Fanuc TP program (LS listing): BOTTOM001.LS

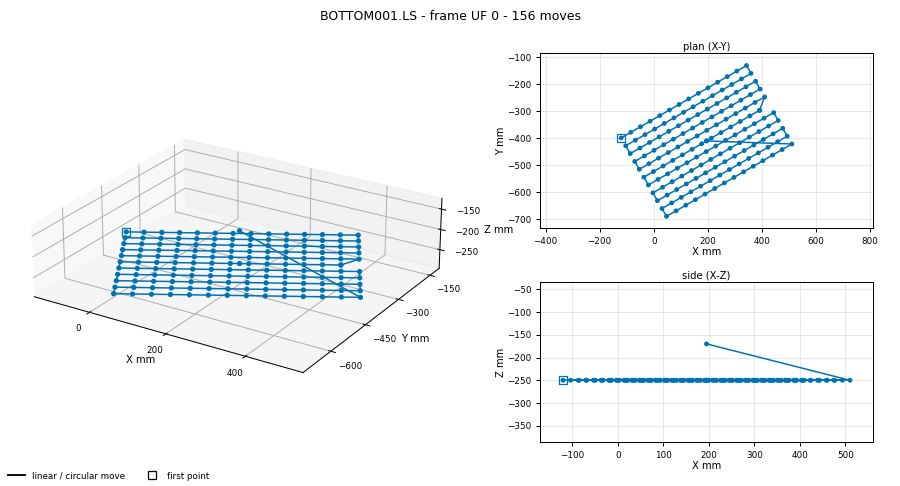
[picture p0: tool path of BOTTOM001.LS in frame UF 0, 156 of 156 moves have a stored position in this frame; points joined in program order, loops and branches not executed]
/PROG  BOTTOM001.LS
/ATTR
OWNER       = MNEDITOR;
COMMENT     = "";
PROG_SIZE   = 636;
CREATE      = DATE 23-01-07  TIME 11:59:14;
MODIFIED    = DATE 23-01-07  TIME 12:02:18;
FILE_NAME   = ;
VERSION     = 0;
LINE_COUNT  = 4;
MEMORY_SIZE = 992;
PROTECT     = READ_WRITE;
TCD:  STACK_SIZE	= 0,
      TASK_PRIORITY	= 50,
      TIME_SLICE	= 0,
      BUSY_LAMP_OFF	= 0,
      ABORT_REQUEST	= 0,
      PAUSE_REQUEST	= 0;
DEFAULT_GROUP	= 1,*,*,*,*;
CONTROL_CODE	= 00000000 00000000;
/MN
   1:J P[1] 100% FINE    ;
   2:L P[2] 100mm/sec CNT0    ;
   3:L P[3] 100mm/sec CNT0    ;
   4:L P[4] 100mm/sec CNT0    ;
   5:L P[5] 100mm/sec CNT0    ;
   6:L P[6] 100mm/sec CNT0    ;
   7:L P[7] 100mm/sec CNT0    ;
   8:L P[8] 100mm/sec CNT0    ;
   9:L P[9] 100mm/sec CNT0    ;
   10:L P[10] 100mm/sec CNT0    ;
   11:L P[11] 100mm/sec CNT0    ;
   12:L P[12] 100mm/sec CNT0    ;
   13:L P[13] 100mm/sec CNT0    ;
   14:L P[14] 100mm/sec CNT0    ;
   15:L P[15] 100mm/sec CNT0    ;
   16:L P[16] 100mm/sec CNT0    ;
   17:L P[17] 100mm/sec CNT0    ;
   18:L P[18] 100mm/sec CNT0    ;
   19:L P[19] 100mm/sec CNT0    ;
   20:L P[20] 100mm/sec CNT0    ;
   21:L P[21] 100mm/sec CNT0    ;
   22:L P[22] 100mm/sec CNT0    ;
   23:L P[23] 100mm/sec CNT0    ;
   24:L P[24] 100mm/sec CNT0    ;
   25:L P[25] 100mm/sec CNT0    ;
   26:L P[26] 100mm/sec CNT0    ;
   27:L P[27] 100mm/sec CNT0    ;
   28:L P[28] 100mm/sec CNT0    ;
   29:L P[29] 100mm/sec CNT0    ;
   30:L P[30] 100mm/sec CNT0    ;
   31:L P[31] 100mm/sec CNT0    ;
   32:L P[32] 100mm/sec CNT0    ;
   33:L P[33] 100mm/sec CNT0    ;
   34:L P[34] 100mm/sec CNT0    ;
   35:L P[35] 100mm/sec CNT0    ;
   36:L P[36] 100mm/sec CNT0    ;
   37:L P[37] 100mm/sec CNT0    ;
   38:L P[38] 100mm/sec CNT0    ;
   39:L P[39] 100mm/sec CNT0    ;
   40:L P[40] 100mm/sec CNT0    ;
   41:L P[41] 100mm/sec CNT0    ;
   42:L P[42] 100mm/sec CNT0    ;
   43:L P[43] 100mm/sec CNT0    ;
   44:L P[44] 100mm/sec CNT0    ;
   45:L P[45] 100mm/sec CNT0    ;
   46:L P[46] 100mm/sec CNT0    ;
   47:L P[47] 100mm/sec CNT0    ;
   48:L P[48] 100mm/sec CNT0    ;
   49:L P[49] 100mm/sec CNT0    ;
   50:L P[50] 100mm/sec CNT0    ;
   51:L P[51] 100mm/sec CNT0    ;
   52:L P[52] 100mm/sec CNT0    ;
   53:L P[53] 100mm/sec CNT0    ;
   54:L P[54] 100mm/sec CNT0    ;
   55:L P[55] 100mm/sec CNT0    ;
   56:L P[56] 100mm/sec CNT0    ;
   57:L P[57] 100mm/sec CNT0    ;
   58:L P[58] 100mm/sec CNT0    ;
   59:L P[59] 100mm/sec CNT0    ;
   60:L P[60] 100mm/sec CNT0    ;
   61:L P[61] 100mm/sec CNT0    ;
   62:L P[62] 100mm/sec CNT0    ;
   63:L P[63] 100mm/sec CNT0    ;
   64:L P[64] 100mm/sec CNT0    ;
   65:L P[65] 100mm/sec CNT0    ;
   66:L P[66] 100mm/sec CNT0    ;
   67:L P[67] 100mm/sec CNT0    ;
   68:L P[68] 100mm/sec CNT0    ;
   69:L P[69] 100mm/sec CNT0    ;
   70:L P[70] 100mm/sec CNT0    ;
   71:L P[71] 100mm/sec CNT0    ;
   72:L P[72] 100mm/sec CNT0    ;
   73:L P[73] 100mm/sec CNT0    ;
   74:L P[74] 100mm/sec CNT0    ;
   75:L P[75] 100mm/sec CNT0    ;
   76:L P[76] 100mm/sec CNT0    ;
   77:L P[77] 100mm/sec CNT0    ;
   78:L P[78] 100mm/sec CNT0    ;
   79:L P[79] 100mm/sec CNT0    ;
   80:L P[80] 100mm/sec CNT0    ;
   81:L P[81] 100mm/sec CNT0    ;
   82:L P[82] 100mm/sec CNT0    ;
   83:L P[83] 100mm/sec CNT0    ;
   84:L P[84] 100mm/sec CNT0    ;
   85:L P[85] 100mm/sec CNT0    ;
   86:L P[86] 100mm/sec CNT0    ;
   87:L P[87] 100mm/sec CNT0    ;
   88:L P[88] 100mm/sec CNT0    ;
   89:L P[89] 100mm/sec CNT0    ;
   90:L P[90] 100mm/sec CNT0    ;
   91:L P[91] 100mm/sec CNT0    ;
   92:L P[92] 100mm/sec CNT0    ;
   93:L P[93] 100mm/sec CNT0    ;
   94:L P[94] 100mm/sec CNT0    ;
   95:L P[95] 100mm/sec CNT0    ;
   96:L P[96] 100mm/sec CNT0    ;
   97:L P[97] 100mm/sec CNT0    ;
   98:L P[98] 100mm/sec CNT0    ;
   99:L P[99] 100mm/sec CNT0    ;
   100:L P[100] 100mm/sec CNT0    ;
   101:L P[101] 100mm/sec CNT0    ;
   102:L P[102] 100mm/sec CNT0    ;
   103:L P[103] 100mm/sec CNT0    ;
   104:L P[104] 100mm/sec CNT0    ;
   105:L P[105] 100mm/sec CNT0    ;
   106:L P[106] 100mm/sec CNT0    ;
   107:L P[107] 100mm/sec CNT0    ;
   108:L P[108] 100mm/sec CNT0    ;
   109:L P[109] 100mm/sec CNT0    ;
   110:L P[110] 100mm/sec CNT0    ;
   111:L P[111] 100mm/sec CNT0    ;
   112:L P[112] 100mm/sec CNT0    ;
   113:L P[113] 100mm/sec CNT0    ;
   114:L P[114] 100mm/sec CNT0    ;
   115:L P[115] 100mm/sec CNT0    ;
   116:L P[116] 100mm/sec CNT0    ;
   117:L P[117] 100mm/sec CNT0    ;
   118:L P[118] 100mm/sec CNT0    ;
   119:L P[119] 100mm/sec CNT0    ;
   120:L P[120] 100mm/sec CNT0    ;
   121:L P[121] 100mm/sec CNT0    ;
   122:L P[122] 100mm/sec CNT0    ;
   123:L P[123] 100mm/sec CNT0    ;
   124:L P[124] 100mm/sec CNT0    ;
   125:L P[125] 100mm/sec CNT0    ;
   126:L P[126] 100mm/sec CNT0    ;
   127:L P[127] 100mm/sec CNT0    ;
   128:L P[128] 100mm/sec CNT0    ;
   129:L P[129] 100mm/sec CNT0    ;
   130:L P[130] 100mm/sec CNT0    ;
   131:L P[131] 100mm/sec CNT0    ;
   132:L P[132] 100mm/sec CNT0    ;
   133:L P[133] 100mm/sec CNT0    ;
   134:L P[134] 100mm/sec CNT0    ;
   135:L P[135] 100mm/sec CNT0    ;
   136:L P[136] 100mm/sec CNT0    ;
   137:L P[137] 100mm/sec CNT0    ;
   138:L P[138] 100mm/sec CNT0    ;
   139:L P[139] 100mm/sec CNT0    ;
   140:L P[140] 100mm/sec CNT0    ;
   141:L P[141] 100mm/sec CNT0    ;
   142:L P[142] 100mm/sec CNT0    ;
   143:L P[143] 100mm/sec CNT0    ;
   144:L P[144] 100mm/sec CNT0    ;
   145:L P[145] 100mm/sec CNT0    ;
   146:L P[146] 100mm/sec CNT0    ;
   147:L P[147] 100mm/sec CNT0    ;
   148:L P[148] 100mm/sec CNT0    ;
   149:L P[149] 100mm/sec CNT0    ;
   150:L P[150] 100mm/sec CNT0    ;
   151:L P[151] 100mm/sec CNT0    ;
   152:L P[152] 100mm/sec CNT0    ;
   153:L P[153] 100mm/sec CNT0    ;
   154:L P[154] 100mm/sec CNT0    ;
   155:L P[155] 100mm/sec CNT0    ;
   156:L P[156] 100mm/sec CNT0    ;
/POS
P[1]{
   GP1:
	UF : 0, UT : 6,		CONFIG : 'N U T, 0, 0, 0',
	X =  -120.438  mm,	Y =   -398.694  mm,	Z =   -250.000  mm,
	W =  90.000 deg,	P =   0.000 deg,	R =   90.000 deg
};
P[2]{
   GP1:
	UF : 0, UT : 6,		CONFIG : 'N U T, 0, 0, 0',
	X =  -84.795  mm,	Y =   -378.115  mm,	Z =   -250.000  mm,
	W =  90.000 deg,	P =   0.000 deg,	R =   90.000 deg
};
P[3]{
   GP1:
	UF : 0, UT : 6,		CONFIG : 'N U T, 0, 0, 0',
	X =  -49.153  mm,	Y =   -357.535  mm,	Z =   -250.000  mm,
	W =  90.000 deg,	P =   0.000 deg,	R =   90.000 deg
};
P[4]{
   GP1:
	UF : 0, UT : 6,		CONFIG : 'N U T, 0, 0, 0',
	X =  -13.511  mm,	Y =   -336.956  mm,	Z =   -250.000  mm,
	W =  90.000 deg,	P =   0.000 deg,	R =   90.000 deg
};
P[5]{
   GP1:
	UF : 0, UT : 6,		CONFIG : 'N U T, 0, 0, 0',
	X =  22.131  mm,	Y =   -316.376  mm,	Z =   -250.000  mm,
	W =  90.000 deg,	P =   0.000 deg,	R =   90.000 deg
};
P[6]{
   GP1:
	UF : 0, UT : 6,		CONFIG : 'N U T, 0, 0, 0',
	X =  57.773  mm,	Y =   -295.797  mm,	Z =   -250.000  mm,
	W =  90.000 deg,	P =   0.000 deg,	R =   90.000 deg
};
P[7]{
   GP1:
	UF : 0, UT : 6,		CONFIG : 'N U T, 0, 0, 0',
	X =  93.415  mm,	Y =   -275.217  mm,	Z =   -250.000  mm,
	W =  90.000 deg,	P =   0.000 deg,	R =   90.000 deg
};
P[8]{
   GP1:
	UF : 0, UT : 6,		CONFIG : 'N U T, 0, 0, 0',
	X =  129.058  mm,	Y =   -254.638  mm,	Z =   -250.000  mm,
	W =  90.000 deg,	P =   0.000 deg,	R =   90.000 deg
};
P[9]{
   GP1:
	UF : 0, UT : 6,		CONFIG : 'N U T, 0, 0, 0',
	X =  164.700  mm,	Y =   -234.059  mm,	Z =   -250.000  mm,
	W =  90.000 deg,	P =   0.000 deg,	R =   90.000 deg
};
P[10]{
   GP1:
	UF : 0, UT : 6,		CONFIG : 'N U T, 0, 0, 0',
	X =  200.342  mm,	Y =   -213.479  mm,	Z =   -250.000  mm,
	W =  90.000 deg,	P =   0.000 deg,	R =   90.000 deg
};
P[11]{
   GP1:
	UF : 0, UT : 6,		CONFIG : 'N U T, 0, 0, 0',
	X =  235.984  mm,	Y =   -192.900  mm,	Z =   -250.000  mm,
	W =  90.000 deg,	P =   0.000 deg,	R =   90.000 deg
};
P[12]{
   GP1:
	UF : 0, UT : 6,		CONFIG : 'N U T, 0, 0, 0',
	X =  271.626  mm,	Y =   -172.320  mm,	Z =   -250.000  mm,
	W =  90.000 deg,	P =   0.000 deg,	R =   90.000 deg
};
P[13]{
   GP1:
	UF : 0, UT : 6,		CONFIG : 'N U T, 0, 0, 0',
	X =  307.268  mm,	Y =   -151.741  mm,	Z =   -250.000  mm,
	W =  90.000 deg,	P =   0.000 deg,	R =   90.000 deg
};
P[14]{
   GP1:
	UF : 0, UT : 6,		CONFIG : 'N U T, 0, 0, 0',
	X =  342.911  mm,	Y =   -131.161  mm,	Z =   -250.000  mm,
	W =  90.000 deg,	P =   0.000 deg,	R =   90.000 deg
};
P[15]{
   GP1:
	UF : 0, UT : 6,		CONFIG : 'N U T, 0, 0, 0',
	X =  359.663  mm,	Y =   -160.176  mm,	Z =   -250.000  mm,
	W =  90.000 deg,	P =   0.000 deg,	R =   90.000 deg
};
P[16]{
   GP1:
	UF : 0, UT : 6,		CONFIG : 'N U T, 0, 0, 0',
	X =  324.021  mm,	Y =   -180.755  mm,	Z =   -250.000  mm,
	W =  90.000 deg,	P =   0.000 deg,	R =   90.000 deg
};
P[17]{
   GP1:
	UF : 0, UT : 6,		CONFIG : 'N U T, 0, 0, 0',
	X =  288.379  mm,	Y =   -201.335  mm,	Z =   -250.000  mm,
	W =  90.000 deg,	P =   0.000 deg,	R =   90.000 deg
};
P[18]{
   GP1:
	UF : 0, UT : 6,		CONFIG : 'N U T, 0, 0, 0',
	X =  252.737  mm,	Y =   -221.914  mm,	Z =   -250.000  mm,
	W =  90.000 deg,	P =   0.000 deg,	R =   90.000 deg
};
P[19]{
   GP1:
	UF : 0, UT : 6,		CONFIG : 'N U T, 0, 0, 0',
	X =  217.095  mm,	Y =   -242.493  mm,	Z =   -250.000  mm,
	W =  90.000 deg,	P =   0.000 deg,	R =   90.000 deg
};
P[20]{
   GP1:
	UF : 0, UT : 6,		CONFIG : 'N U T, 0, 0, 0',
	X =  181.452  mm,	Y =   -263.073  mm,	Z =   -250.000  mm,
	W =  90.000 deg,	P =   0.000 deg,	R =   90.000 deg
};
P[21]{
   GP1:
	UF : 0, UT : 6,		CONFIG : 'N U T, 0, 0, 0',
	X =  145.810  mm,	Y =   -283.652  mm,	Z =   -250.000  mm,
	W =  90.000 deg,	P =   0.000 deg,	R =   90.000 deg
};
P[22]{
   GP1:
	UF : 0, UT : 6,		CONFIG : 'N U T, 0, 0, 0',
	X =  110.168  mm,	Y =   -304.232  mm,	Z =   -250.000  mm,
	W =  90.000 deg,	P =   0.000 deg,	R =   90.000 deg
};
P[23]{
   GP1:
	UF : 0, UT : 6,		CONFIG : 'N U T, 0, 0, 0',
	X =  74.526  mm,	Y =   -324.811  mm,	Z =   -250.000  mm,
	W =  90.000 deg,	P =   0.000 deg,	R =   90.000 deg
};
P[24]{
   GP1:
	UF : 0, UT : 6,		CONFIG : 'N U T, 0, 0, 0',
	X =  38.884  mm,	Y =   -345.391  mm,	Z =   -250.000  mm,
	W =  90.000 deg,	P =   0.000 deg,	R =   90.000 deg
};
P[25]{
   GP1:
	UF : 0, UT : 6,		CONFIG : 'N U T, 0, 0, 0',
	X =  3.242  mm,	Y =   -365.970  mm,	Z =   -250.000  mm,
	W =  90.000 deg,	P =   0.000 deg,	R =   90.000 deg
};
P[26]{
   GP1:
	UF : 0, UT : 6,		CONFIG : 'N U T, 0, 0, 0',
	X =  -32.401  mm,	Y =   -386.550  mm,	Z =   -250.000  mm,
	W =  90.000 deg,	P =   0.000 deg,	R =   90.000 deg
};
P[27]{
   GP1:
	UF : 0, UT : 6,		CONFIG : 'N U T, 0, 0, 0',
	X =  -68.043  mm,	Y =   -407.129  mm,	Z =   -250.000  mm,
	W =  90.000 deg,	P =   0.000 deg,	R =   90.000 deg
};
P[28]{
   GP1:
	UF : 0, UT : 6,		CONFIG : 'N U T, 0, 0, 0',
	X =  -103.685  mm,	Y =   -427.709  mm,	Z =   -250.000  mm,
	W =  90.000 deg,	P =   0.000 deg,	R =   90.000 deg
};
P[29]{
   GP1:
	UF : 0, UT : 6,		CONFIG : 'N U T, 0, 0, 0',
	X =  -86.932  mm,	Y =   -456.723  mm,	Z =   -250.000  mm,
	W =  90.000 deg,	P =   0.000 deg,	R =   90.000 deg
};
P[30]{
   GP1:
	UF : 0, UT : 6,		CONFIG : 'N U T, 0, 0, 0',
	X =  -51.290  mm,	Y =   -436.144  mm,	Z =   -250.000  mm,
	W =  90.000 deg,	P =   0.000 deg,	R =   90.000 deg
};
P[31]{
   GP1:
	UF : 0, UT : 6,		CONFIG : 'N U T, 0, 0, 0',
	X =  -15.648  mm,	Y =   -415.564  mm,	Z =   -250.000  mm,
	W =  90.000 deg,	P =   0.000 deg,	R =   90.000 deg
};
P[32]{
   GP1:
	UF : 0, UT : 6,		CONFIG : 'N U T, 0, 0, 0',
	X =  19.994  mm,	Y =   -394.985  mm,	Z =   -250.000  mm,
	W =  90.000 deg,	P =   0.000 deg,	R =   90.000 deg
};
P[33]{
   GP1:
	UF : 0, UT : 6,		CONFIG : 'N U T, 0, 0, 0',
	X =  55.636  mm,	Y =   -374.405  mm,	Z =   -250.000  mm,
	W =  90.000 deg,	P =   0.000 deg,	R =   90.000 deg
};
P[34]{
   GP1:
	UF : 0, UT : 6,		CONFIG : 'N U T, 0, 0, 0',
	X =  91.279  mm,	Y =   -353.826  mm,	Z =   -250.000  mm,
	W =  90.000 deg,	P =   0.000 deg,	R =   90.000 deg
};
P[35]{
   GP1:
	UF : 0, UT : 6,		CONFIG : 'N U T, 0, 0, 0',
	X =  126.921  mm,	Y =   -333.246  mm,	Z =   -250.000  mm,
	W =  90.000 deg,	P =   0.000 deg,	R =   90.000 deg
};
P[36]{
   GP1:
	UF : 0, UT : 6,		CONFIG : 'N U T, 0, 0, 0',
	X =  162.563  mm,	Y =   -312.667  mm,	Z =   -250.000  mm,
	W =  90.000 deg,	P =   0.000 deg,	R =   90.000 deg
};
P[37]{
   GP1:
	UF : 0, UT : 6,		CONFIG : 'N U T, 0, 0, 0',
	X =  198.205  mm,	Y =   -292.087  mm,	Z =   -250.000  mm,
	W =  90.000 deg,	P =   0.000 deg,	R =   90.000 deg
};
P[38]{
   GP1:
	UF : 0, UT : 6,		CONFIG : 'N U T, 0, 0, 0',
	X =  233.847  mm,	Y =   -271.508  mm,	Z =   -250.000  mm,
	W =  90.000 deg,	P =   0.000 deg,	R =   90.000 deg
};
P[39]{
   GP1:
	UF : 0, UT : 6,		CONFIG : 'N U T, 0, 0, 0',
	X =  269.490  mm,	Y =   -250.928  mm,	Z =   -250.000  mm,
	W =  90.000 deg,	P =   0.000 deg,	R =   90.000 deg
};
P[40]{
   GP1:
	UF : 0, UT : 6,		CONFIG : 'N U T, 0, 0, 0',
	X =  305.132  mm,	Y =   -230.349  mm,	Z =   -250.000  mm,
	W =  90.000 deg,	P =   0.000 deg,	R =   90.000 deg
};
P[41]{
   GP1:
	UF : 0, UT : 6,		CONFIG : 'N U T, 0, 0, 0',
	X =  340.774  mm,	Y =   -209.769  mm,	Z =   -250.000  mm,
	W =  90.000 deg,	P =   0.000 deg,	R =   90.000 deg
};
P[42]{
   GP1:
	UF : 0, UT : 6,		CONFIG : 'N U T, 0, 0, 0',
	X =  376.416  mm,	Y =   -189.190  mm,	Z =   -250.000  mm,
	W =  90.000 deg,	P =   0.000 deg,	R =   90.000 deg
};
P[43]{
   GP1:
	UF : 0, UT : 6,		CONFIG : 'N U T, 0, 0, 0',
	X =  393.169  mm,	Y =   -218.204  mm,	Z =   -250.000  mm,
	W =  90.000 deg,	P =   0.000 deg,	R =   90.000 deg
};
P[44]{
   GP1:
	UF : 0, UT : 6,		CONFIG : 'N U T, 0, 0, 0',
	X =  357.527  mm,	Y =   -238.784  mm,	Z =   -250.000  mm,
	W =  90.000 deg,	P =   0.000 deg,	R =   90.000 deg
};
P[45]{
   GP1:
	UF : 0, UT : 6,		CONFIG : 'N U T, 0, 0, 0',
	X =  321.884  mm,	Y =   -259.363  mm,	Z =   -250.000  mm,
	W =  90.000 deg,	P =   0.000 deg,	R =   90.000 deg
};
P[46]{
   GP1:
	UF : 0, UT : 6,		CONFIG : 'N U T, 0, 0, 0',
	X =  286.242  mm,	Y =   -279.943  mm,	Z =   -250.000  mm,
	W =  90.000 deg,	P =   0.000 deg,	R =   90.000 deg
};
P[47]{
   GP1:
	UF : 0, UT : 6,		CONFIG : 'N U T, 0, 0, 0',
	X =  250.600  mm,	Y =   -300.522  mm,	Z =   -250.000  mm,
	W =  90.000 deg,	P =   0.000 deg,	R =   90.000 deg
};
P[48]{
   GP1:
	UF : 0, UT : 6,		CONFIG : 'N U T, 0, 0, 0',
	X =  214.958  mm,	Y =   -321.102  mm,	Z =   -250.000  mm,
	W =  90.000 deg,	P =   0.000 deg,	R =   90.000 deg
};
P[49]{
   GP1:
	UF : 0, UT : 6,		CONFIG : 'N U T, 0, 0, 0',
	X =  179.316  mm,	Y =   -341.681  mm,	Z =   -250.000  mm,
	W =  90.000 deg,	P =   0.000 deg,	R =   90.000 deg
};
P[50]{
   GP1:
	UF : 0, UT : 6,		CONFIG : 'N U T, 0, 0, 0',
	X =  143.674  mm,	Y =   -362.261  mm,	Z =   -250.000  mm,
	W =  90.000 deg,	P =   0.000 deg,	R =   90.000 deg
};
P[51]{
   GP1:
	UF : 0, UT : 6,		CONFIG : 'N U T, 0, 0, 0',
	X =  108.031  mm,	Y =   -382.840  mm,	Z =   -250.000  mm,
	W =  90.000 deg,	P =   0.000 deg,	R =   90.000 deg
};
P[52]{
   GP1:
	UF : 0, UT : 6,		CONFIG : 'N U T, 0, 0, 0',
	X =  72.389  mm,	Y =   -403.420  mm,	Z =   -250.000  mm,
	W =  90.000 deg,	P =   0.000 deg,	R =   90.000 deg
};
P[53]{
   GP1:
	UF : 0, UT : 6,		CONFIG : 'N U T, 0, 0, 0',
	X =  36.747  mm,	Y =   -423.999  mm,	Z =   -250.000  mm,
	W =  90.000 deg,	P =   0.000 deg,	R =   90.000 deg
};
P[54]{
   GP1:
	UF : 0, UT : 6,		CONFIG : 'N U T, 0, 0, 0',
	X =  1.105  mm,	Y =   -444.579  mm,	Z =   -250.000  mm,
	W =  90.000 deg,	P =   0.000 deg,	R =   90.000 deg
};
P[55]{
   GP1:
	UF : 0, UT : 6,		CONFIG : 'N U T, 0, 0, 0',
	X =  -34.537  mm,	Y =   -465.158  mm,	Z =   -250.000  mm,
	W =  90.000 deg,	P =   0.000 deg,	R =   90.000 deg
};
P[56]{
   GP1:
	UF : 0, UT : 6,		CONFIG : 'N U T, 0, 0, 0',
	X =  -70.180  mm,	Y =   -485.738  mm,	Z =   -250.000  mm,
	W =  90.000 deg,	P =   0.000 deg,	R =   90.000 deg
};
P[57]{
   GP1:
	UF : 0, UT : 6,		CONFIG : 'N U T, 0, 0, 0',
	X =  -53.427  mm,	Y =   -514.752  mm,	Z =   -250.000  mm,
	W =  90.000 deg,	P =   0.000 deg,	R =   90.000 deg
};
P[58]{
   GP1:
	UF : 0, UT : 6,		CONFIG : 'N U T, 0, 0, 0',
	X =  -17.785  mm,	Y =   -494.173  mm,	Z =   -250.000  mm,
	W =  90.000 deg,	P =   0.000 deg,	R =   90.000 deg
};
P[59]{
   GP1:
	UF : 0, UT : 6,		CONFIG : 'N U T, 0, 0, 0',
	X =  17.858  mm,	Y =   -473.593  mm,	Z =   -250.000  mm,
	W =  90.000 deg,	P =   0.000 deg,	R =   90.000 deg
};
P[60]{
   GP1:
	UF : 0, UT : 6,		CONFIG : 'N U T, 0, 0, 0',
	X =  53.500  mm,	Y =   -453.014  mm,	Z =   -250.000  mm,
	W =  90.000 deg,	P =   0.000 deg,	R =   90.000 deg
};
P[61]{
   GP1:
	UF : 0, UT : 6,		CONFIG : 'N U T, 0, 0, 0',
	X =  89.142  mm,	Y =   -432.434  mm,	Z =   -250.000  mm,
	W =  90.000 deg,	P =   0.000 deg,	R =   90.000 deg
};
P[62]{
   GP1:
	UF : 0, UT : 6,		CONFIG : 'N U T, 0, 0, 0',
	X =  124.784  mm,	Y =   -411.855  mm,	Z =   -250.000  mm,
	W =  90.000 deg,	P =   0.000 deg,	R =   90.000 deg
};
P[63]{
   GP1:
	UF : 0, UT : 6,		CONFIG : 'N U T, 0, 0, 0',
	X =  160.426  mm,	Y =   -391.275  mm,	Z =   -250.000  mm,
	W =  90.000 deg,	P =   0.000 deg,	R =   90.000 deg
};
P[64]{
   GP1:
	UF : 0, UT : 6,		CONFIG : 'N U T, 0, 0, 0',
	X =  196.068  mm,	Y =   -370.696  mm,	Z =   -250.000  mm,
	W =  90.000 deg,	P =   0.000 deg,	R =   90.000 deg
};
P[65]{
   GP1:
	UF : 0, UT : 6,		CONFIG : 'N U T, 0, 0, 0',
	X =  231.711  mm,	Y =   -350.116  mm,	Z =   -250.000  mm,
	W =  90.000 deg,	P =   0.000 deg,	R =   90.000 deg
};
P[66]{
   GP1:
	UF : 0, UT : 6,		CONFIG : 'N U T, 0, 0, 0',
	X =  267.353  mm,	Y =   -329.537  mm,	Z =   -250.000  mm,
	W =  90.000 deg,	P =   0.000 deg,	R =   90.000 deg
};
P[67]{
   GP1:
	UF : 0, UT : 6,		CONFIG : 'N U T, 0, 0, 0',
	X =  302.995  mm,	Y =   -308.957  mm,	Z =   -250.000  mm,
	W =  90.000 deg,	P =   0.000 deg,	R =   90.000 deg
};
P[68]{
   GP1:
	UF : 0, UT : 6,		CONFIG : 'N U T, 0, 0, 0',
	X =  338.637  mm,	Y =   -288.378  mm,	Z =   -250.000  mm,
	W =  90.000 deg,	P =   0.000 deg,	R =   90.000 deg
};
P[69]{
   GP1:
	UF : 0, UT : 6,		CONFIG : 'N U T, 0, 0, 0',
	X =  374.279  mm,	Y =   -267.798  mm,	Z =   -250.000  mm,
	W =  90.000 deg,	P =   0.000 deg,	R =   90.000 deg
};
P[70]{
   GP1:
	UF : 0, UT : 6,		CONFIG : 'N U T, 0, 0, 0',
	X =  409.921  mm,	Y =   -247.219  mm,	Z =   -250.000  mm,
	W =  90.000 deg,	P =   0.000 deg,	R =   90.000 deg
};
P[71]{
   GP1:
	UF : 0, UT : 6,		CONFIG : 'N U T, 0, 0, 0',
	X =  391.032  mm,	Y =   -296.813  mm,	Z =   -250.000  mm,
	W =  90.000 deg,	P =   0.000 deg,	R =   90.000 deg
};
P[72]{
   GP1:
	UF : 0, UT : 6,		CONFIG : 'N U T, 0, 0, 0',
	X =  391.032  mm,	Y =   -296.813  mm,	Z =   -250.000  mm,
	W =  90.000 deg,	P =   0.000 deg,	R =   90.000 deg
};
P[73]{
   GP1:
	UF : 0, UT : 6,		CONFIG : 'N U T, 0, 0, 0',
	X =  355.390  mm,	Y =   -317.392  mm,	Z =   -250.000  mm,
	W =  90.000 deg,	P =   0.000 deg,	R =   90.000 deg
};
P[74]{
   GP1:
	UF : 0, UT : 6,		CONFIG : 'N U T, 0, 0, 0',
	X =  319.748  mm,	Y =   -337.972  mm,	Z =   -250.000  mm,
	W =  90.000 deg,	P =   0.000 deg,	R =   90.000 deg
};
P[75]{
   GP1:
	UF : 0, UT : 6,		CONFIG : 'N U T, 0, 0, 0',
	X =  284.105  mm,	Y =   -358.551  mm,	Z =   -250.000  mm,
	W =  90.000 deg,	P =   0.000 deg,	R =   90.000 deg
};
P[76]{
   GP1:
	UF : 0, UT : 6,		CONFIG : 'N U T, 0, 0, 0',
	X =  248.463  mm,	Y =   -379.131  mm,	Z =   -250.000  mm,
	W =  90.000 deg,	P =   0.000 deg,	R =   90.000 deg
};
P[77]{
   GP1:
	UF : 0, UT : 6,		CONFIG : 'N U T, 0, 0, 0',
	X =  212.821  mm,	Y =   -399.710  mm,	Z =   -250.000  mm,
	W =  90.000 deg,	P =   0.000 deg,	R =   90.000 deg
};
P[78]{
   GP1:
	UF : 0, UT : 6,		CONFIG : 'N U T, 0, 0, 0',
	X =  195.000  mm,	Y =   -410.000  mm,	Z =   -250.000  mm,
	W =  90.000 deg,	P =   0.000 deg,	R =   90.000 deg
};
P[79]{
   GP1:
	UF : 0, UT : 6,		CONFIG : 'N U T, 0, 0, 0',
	X =  177.179  mm,	Y =   -420.290  mm,	Z =   -250.000  mm,
	W =  90.000 deg,	P =   0.000 deg,	R =   90.000 deg
};
P[80]{
   GP1:
	UF : 0, UT : 6,		CONFIG : 'N U T, 0, 0, 0',
	X =  141.537  mm,	Y =   -440.869  mm,	Z =   -250.000  mm,
	W =  90.000 deg,	P =   0.000 deg,	R =   90.000 deg
};
P[81]{
   GP1:
	UF : 0, UT : 6,		CONFIG : 'N U T, 0, 0, 0',
	X =  105.895  mm,	Y =   -461.449  mm,	Z =   -250.000  mm,
	W =  90.000 deg,	P =   0.000 deg,	R =   90.000 deg
};
P[82]{
   GP1:
	UF : 0, UT : 6,		CONFIG : 'N U T, 0, 0, 0',
	X =  70.252  mm,	Y =   -482.028  mm,	Z =   -250.000  mm,
	W =  90.000 deg,	P =   0.000 deg,	R =   90.000 deg
};
P[83]{
   GP1:
	UF : 0, UT : 6,		CONFIG : 'N U T, 0, 0, 0',
	X =  34.610  mm,	Y =   -502.608  mm,	Z =   -250.000  mm,
	W =  90.000 deg,	P =   0.000 deg,	R =   90.000 deg
};
P[84]{
   GP1:
	UF : 0, UT : 6,		CONFIG : 'N U T, 0, 0, 0',
	X =  -1.032  mm,	Y =   -523.187  mm,	Z =   -250.000  mm,
	W =  90.000 deg,	P =   0.000 deg,	R =   90.000 deg
};
P[85]{
   GP1:
	UF : 0, UT : 6,		CONFIG : 'N U T, 0, 0, 0',
	X =  -36.674  mm,	Y =   -543.767  mm,	Z =   -250.000  mm,
	W =  90.000 deg,	P =   0.000 deg,	R =   90.000 deg
};
P[86]{
   GP1:
	UF : 0, UT : 6,		CONFIG : 'N U T, 0, 0, 0',
	X =  -19.921  mm,	Y =   -572.781  mm,	Z =   -250.000  mm,
	W =  90.000 deg,	P =   0.000 deg,	R =   90.000 deg
};
P[87]{
   GP1:
	UF : 0, UT : 6,		CONFIG : 'N U T, 0, 0, 0',
	X =  15.721  mm,	Y =   -552.202  mm,	Z =   -250.000  mm,
	W =  90.000 deg,	P =   0.000 deg,	R =   90.000 deg
};
P[88]{
   GP1:
	UF : 0, UT : 6,		CONFIG : 'N U T, 0, 0, 0',
	X =  51.363  mm,	Y =   -531.622  mm,	Z =   -250.000  mm,
	W =  90.000 deg,	P =   0.000 deg,	R =   90.000 deg
};
P[89]{
   GP1:
	UF : 0, UT : 6,		CONFIG : 'N U T, 0, 0, 0',
	X =  87.005  mm,	Y =   -511.043  mm,	Z =   -250.000  mm,
	W =  90.000 deg,	P =   0.000 deg,	R =   90.000 deg
};
P[90]{
   GP1:
	UF : 0, UT : 6,		CONFIG : 'N U T, 0, 0, 0',
	X =  122.647  mm,	Y =   -490.463  mm,	Z =   -250.000  mm,
	W =  90.000 deg,	P =   0.000 deg,	R =   90.000 deg
};
P[91]{
   GP1:
	UF : 0, UT : 6,		CONFIG : 'N U T, 0, 0, 0',
	X =  158.289  mm,	Y =   -469.884  mm,	Z =   -250.000  mm,
	W =  90.000 deg,	P =   0.000 deg,	R =   90.000 deg
};
P[92]{
   GP1:
	UF : 0, UT : 6,		CONFIG : 'N U T, 0, 0, 0',
	X =  193.932  mm,	Y =   -449.304  mm,	Z =   -250.000  mm,
	W =  90.000 deg,	P =   0.000 deg,	R =   90.000 deg
};
P[93]{
   GP1:
	UF : 0, UT : 6,		CONFIG : 'N U T, 0, 0, 0',
	X =  229.574  mm,	Y =   -428.725  mm,	Z =   -250.000  mm,
	W =  90.000 deg,	P =   0.000 deg,	R =   90.000 deg
};
P[94]{
   GP1:
	UF : 0, UT : 6,		CONFIG : 'N U T, 0, 0, 0',
	X =  265.216  mm,	Y =   -408.145  mm,	Z =   -250.000  mm,
	W =  90.000 deg,	P =   0.000 deg,	R =   90.000 deg
};
P[95]{
   GP1:
	UF : 0, UT : 6,		CONFIG : 'N U T, 0, 0, 0',
	X =  300.858  mm,	Y =   -387.566  mm,	Z =   -250.000  mm,
	W =  90.000 deg,	P =   0.000 deg,	R =   90.000 deg
};
P[96]{
   GP1:
	UF : 0, UT : 6,		CONFIG : 'N U T, 0, 0, 0',
	X =  336.500  mm,	Y =   -366.986  mm,	Z =   -250.000  mm,
	W =  90.000 deg,	P =   0.000 deg,	R =   90.000 deg
};
P[97]{
   GP1:
	UF : 0, UT : 6,		CONFIG : 'N U T, 0, 0, 0',
	X =  372.142  mm,	Y =   -346.407  mm,	Z =   -250.000  mm,
	W =  90.000 deg,	P =   0.000 deg,	R =   90.000 deg
};
P[98]{
   GP1:
	UF : 0, UT : 6,		CONFIG : 'N U T, 0, 0, 0',
	X =  407.785  mm,	Y =   -325.827  mm,	Z =   -250.000  mm,
	W =  90.000 deg,	P =   0.000 deg,	R =   90.000 deg
};
P[99]{
   GP1:
	UF : 0, UT : 6,		CONFIG : 'N U T, 0, 0, 0',
	X =  443.427  mm,	Y =   -305.248  mm,	Z =   -250.000  mm,
	W =  90.000 deg,	P =   0.000 deg,	R =   90.000 deg
};
P[100]{
   GP1:
	UF : 0, UT : 6,		CONFIG : 'N U T, 0, 0, 0',
	X =  460.180  mm,	Y =   -334.262  mm,	Z =   -250.000  mm,
	W =  90.000 deg,	P =   0.000 deg,	R =   90.000 deg
};
P[101]{
   GP1:
	UF : 0, UT : 6,		CONFIG : 'N U T, 0, 0, 0',
	X =  424.537  mm,	Y =   -354.842  mm,	Z =   -250.000  mm,
	W =  90.000 deg,	P =   0.000 deg,	R =   90.000 deg
};
P[102]{
   GP1:
	UF : 0, UT : 6,		CONFIG : 'N U T, 0, 0, 0',
	X =  388.895  mm,	Y =   -375.421  mm,	Z =   -250.000  mm,
	W =  90.000 deg,	P =   0.000 deg,	R =   90.000 deg
};
P[103]{
   GP1:
	UF : 0, UT : 6,		CONFIG : 'N U T, 0, 0, 0',
	X =  353.253  mm,	Y =   -396.001  mm,	Z =   -250.000  mm,
	W =  90.000 deg,	P =   0.000 deg,	R =   90.000 deg
};
P[104]{
   GP1:
	UF : 0, UT : 6,		CONFIG : 'N U T, 0, 0, 0',
	X =  317.611  mm,	Y =   -416.580  mm,	Z =   -250.000  mm,
	W =  90.000 deg,	P =   0.000 deg,	R =   90.000 deg
};
P[105]{
   GP1:
	UF : 0, UT : 6,		CONFIG : 'N U T, 0, 0, 0',
	X =  281.969  mm,	Y =   -437.160  mm,	Z =   -250.000  mm,
	W =  90.000 deg,	P =   0.000 deg,	R =   90.000 deg
};
P[106]{
   GP1:
	UF : 0, UT : 6,		CONFIG : 'N U T, 0, 0, 0',
	X =  246.326  mm,	Y =   -457.739  mm,	Z =   -250.000  mm,
	W =  90.000 deg,	P =   0.000 deg,	R =   90.000 deg
};
P[107]{
   GP1:
	UF : 0, UT : 6,		CONFIG : 'N U T, 0, 0, 0',
	X =  210.684  mm,	Y =   -478.319  mm,	Z =   -250.000  mm,
	W =  90.000 deg,	P =   0.000 deg,	R =   90.000 deg
};
P[108]{
   GP1:
	UF : 0, UT : 6,		CONFIG : 'N U T, 0, 0, 0',
	X =  175.042  mm,	Y =   -498.898  mm,	Z =   -250.000  mm,
	W =  90.000 deg,	P =   0.000 deg,	R =   90.000 deg
};
P[109]{
   GP1:
	UF : 0, UT : 6,		CONFIG : 'N U T, 0, 0, 0',
	X =  139.400  mm,	Y =   -519.478  mm,	Z =   -250.000  mm,
	W =  90.000 deg,	P =   0.000 deg,	R =   90.000 deg
};
P[110]{
   GP1:
	UF : 0, UT : 6,		CONFIG : 'N U T, 0, 0, 0',
	X =  103.758  mm,	Y =   -540.057  mm,	Z =   -250.000  mm,
	W =  90.000 deg,	P =   0.000 deg,	R =   90.000 deg
};
P[111]{
   GP1:
	UF : 0, UT : 6,		CONFIG : 'N U T, 0, 0, 0',
	X =  68.116  mm,	Y =   -560.637  mm,	Z =   -250.000  mm,
	W =  90.000 deg,	P =   0.000 deg,	R =   90.000 deg
};
P[112]{
   GP1:
	UF : 0, UT : 6,		CONFIG : 'N U T, 0, 0, 0',
	X =  32.473  mm,	Y =   -581.216  mm,	Z =   -250.000  mm,
	W =  90.000 deg,	P =   0.000 deg,	R =   90.000 deg
};
P[113]{
   GP1:
	UF : 0, UT : 6,		CONFIG : 'N U T, 0, 0, 0',
	X =  -3.169  mm,	Y =   -601.796  mm,	Z =   -250.000  mm,
	W =  90.000 deg,	P =   0.000 deg,	R =   90.000 deg
};
P[114]{
   GP1:
	UF : 0, UT : 6,		CONFIG : 'N U T, 0, 0, 0',
	X =  13.584  mm,	Y =   -630.810  mm,	Z =   -250.000  mm,
	W =  90.000 deg,	P =   0.000 deg,	R =   90.000 deg
};
P[115]{
   GP1:
	UF : 0, UT : 6,		CONFIG : 'N U T, 0, 0, 0',
	X =  49.226  mm,	Y =   -610.231  mm,	Z =   -250.000  mm,
	W =  90.000 deg,	P =   0.000 deg,	R =   90.000 deg
};
P[116]{
   GP1:
	UF : 0, UT : 6,		CONFIG : 'N U T, 0, 0, 0',
	X =  84.868  mm,	Y =   -589.651  mm,	Z =   -250.000  mm,
	W =  90.000 deg,	P =   0.000 deg,	R =   90.000 deg
};
P[117]{
   GP1:
	UF : 0, UT : 6,		CONFIG : 'N U T, 0, 0, 0',
	X =  120.510  mm,	Y =   -569.072  mm,	Z =   -250.000  mm,
	W =  90.000 deg,	P =   0.000 deg,	R =   90.000 deg
};
P[118]{
   GP1:
	UF : 0, UT : 6,		CONFIG : 'N U T, 0, 0, 0',
	X =  156.153  mm,	Y =   -548.492  mm,	Z =   -250.000  mm,
	W =  90.000 deg,	P =   0.000 deg,	R =   90.000 deg
};
P[119]{
   GP1:
	UF : 0, UT : 6,		CONFIG : 'N U T, 0, 0, 0',
	X =  191.795  mm,	Y =   -527.913  mm,	Z =   -250.000  mm,
	W =  90.000 deg,	P =   0.000 deg,	R =   90.000 deg
};
P[120]{
   GP1:
	UF : 0, UT : 6,		CONFIG : 'N U T, 0, 0, 0',
	X =  227.437  mm,	Y =   -507.333  mm,	Z =   -250.000  mm,
	W =  90.000 deg,	P =   0.000 deg,	R =   90.000 deg
};
P[121]{
   GP1:
	UF : 0, UT : 6,		CONFIG : 'N U T, 0, 0, 0',
	X =  263.079  mm,	Y =   -486.754  mm,	Z =   -250.000  mm,
	W =  90.000 deg,	P =   0.000 deg,	R =   90.000 deg
};
P[122]{
   GP1:
	UF : 0, UT : 6,		CONFIG : 'N U T, 0, 0, 0',
	X =  298.721  mm,	Y =   -466.174  mm,	Z =   -250.000  mm,
	W =  90.000 deg,	P =   0.000 deg,	R =   90.000 deg
};
P[123]{
   GP1:
	UF : 0, UT : 6,		CONFIG : 'N U T, 0, 0, 0',
	X =  334.364  mm,	Y =   -445.595  mm,	Z =   -250.000  mm,
	W =  90.000 deg,	P =   0.000 deg,	R =   90.000 deg
};
P[124]{
   GP1:
	UF : 0, UT : 6,		CONFIG : 'N U T, 0, 0, 0',
	X =  370.006  mm,	Y =   -425.015  mm,	Z =   -250.000  mm,
	W =  90.000 deg,	P =   0.000 deg,	R =   90.000 deg
};
P[125]{
   GP1:
	UF : 0, UT : 6,		CONFIG : 'N U T, 0, 0, 0',
	X =  405.648  mm,	Y =   -404.436  mm,	Z =   -250.000  mm,
	W =  90.000 deg,	P =   0.000 deg,	R =   90.000 deg
};
P[126]{
   GP1:
	UF : 0, UT : 6,		CONFIG : 'N U T, 0, 0, 0',
	X =  441.290  mm,	Y =   -383.856  mm,	Z =   -250.000  mm,
	W =  90.000 deg,	P =   0.000 deg,	R =   90.000 deg
};
P[127]{
   GP1:
	UF : 0, UT : 6,		CONFIG : 'N U T, 0, 0, 0',
	X =  476.932  mm,	Y =   -363.277  mm,	Z =   -250.000  mm,
	W =  90.000 deg,	P =   0.000 deg,	R =   90.000 deg
};
P[128]{
   GP1:
	UF : 0, UT : 6,		CONFIG : 'N U T, 0, 0, 0',
	X =  493.685  mm,	Y =   -392.291  mm,	Z =   -250.000  mm,
	W =  90.000 deg,	P =   0.000 deg,	R =   90.000 deg
};
P[129]{
   GP1:
	UF : 0, UT : 6,		CONFIG : 'N U T, 0, 0, 0',
	X =  458.043  mm,	Y =   -412.871  mm,	Z =   -250.000  mm,
	W =  90.000 deg,	P =   0.000 deg,	R =   90.000 deg
};
P[130]{
   GP1:
	UF : 0, UT : 6,		CONFIG : 'N U T, 0, 0, 0',
	X =  422.401  mm,	Y =   -433.450  mm,	Z =   -250.000  mm,
	W =  90.000 deg,	P =   0.000 deg,	R =   90.000 deg
};
P[131]{
   GP1:
	UF : 0, UT : 6,		CONFIG : 'N U T, 0, 0, 0',
	X =  386.758  mm,	Y =   -454.030  mm,	Z =   -250.000  mm,
	W =  90.000 deg,	P =   0.000 deg,	R =   90.000 deg
};
P[132]{
   GP1:
	UF : 0, UT : 6,		CONFIG : 'N U T, 0, 0, 0',
	X =  351.116  mm,	Y =   -474.609  mm,	Z =   -250.000  mm,
	W =  90.000 deg,	P =   0.000 deg,	R =   90.000 deg
};
P[133]{
   GP1:
	UF : 0, UT : 6,		CONFIG : 'N U T, 0, 0, 0',
	X =  315.474  mm,	Y =   -495.189  mm,	Z =   -250.000  mm,
	W =  90.000 deg,	P =   0.000 deg,	R =   90.000 deg
};
P[134]{
   GP1:
	UF : 0, UT : 6,		CONFIG : 'N U T, 0, 0, 0',
	X =  279.832  mm,	Y =   -515.768  mm,	Z =   -250.000  mm,
	W =  90.000 deg,	P =   0.000 deg,	R =   90.000 deg
};
P[135]{
   GP1:
	UF : 0, UT : 6,		CONFIG : 'N U T, 0, 0, 0',
	X =  244.190  mm,	Y =   -536.348  mm,	Z =   -250.000  mm,
	W =  90.000 deg,	P =   0.000 deg,	R =   90.000 deg
};
P[136]{
   GP1:
	UF : 0, UT : 6,		CONFIG : 'N U T, 0, 0, 0',
	X =  208.548  mm,	Y =   -556.927  mm,	Z =   -250.000  mm,
	W =  90.000 deg,	P =   0.000 deg,	R =   90.000 deg
};
P[137]{
   GP1:
	UF : 0, UT : 6,		CONFIG : 'N U T, 0, 0, 0',
	X =  172.905  mm,	Y =   -577.507  mm,	Z =   -250.000  mm,
	W =  90.000 deg,	P =   0.000 deg,	R =   90.000 deg
};
P[138]{
   GP1:
	UF : 0, UT : 6,		CONFIG : 'N U T, 0, 0, 0',
	X =  137.263  mm,	Y =   -598.086  mm,	Z =   -250.000  mm,
	W =  90.000 deg,	P =   0.000 deg,	R =   90.000 deg
};
P[139]{
   GP1:
	UF : 0, UT : 6,		CONFIG : 'N U T, 0, 0, 0',
	X =  101.621  mm,	Y =   -618.665  mm,	Z =   -250.000  mm,
	W =  90.000 deg,	P =   0.000 deg,	R =   90.000 deg
};
P[140]{
   GP1:
	UF : 0, UT : 6,		CONFIG : 'N U T, 0, 0, 0',
	X =  65.979  mm,	Y =   -639.245  mm,	Z =   -250.000  mm,
	W =  90.000 deg,	P =   0.000 deg,	R =   90.000 deg
};
P[141]{
   GP1:
	UF : 0, UT : 6,		CONFIG : 'N U T, 0, 0, 0',
	X =  30.337  mm,	Y =   -659.824  mm,	Z =   -250.000  mm,
	W =  90.000 deg,	P =   0.000 deg,	R =   90.000 deg
};
P[142]{
   GP1:
	UF : 0, UT : 6,		CONFIG : 'N U T, 0, 0, 0',
	X =  47.089  mm,	Y =   -688.839  mm,	Z =   -250.000  mm,
	W =  90.000 deg,	P =   0.000 deg,	R =   90.000 deg
};
P[143]{
   GP1:
	UF : 0, UT : 6,		CONFIG : 'N U T, 0, 0, 0',
	X =  82.732  mm,	Y =   -668.259  mm,	Z =   -250.000  mm,
	W =  90.000 deg,	P =   0.000 deg,	R =   90.000 deg
};
P[144]{
   GP1:
	UF : 0, UT : 6,		CONFIG : 'N U T, 0, 0, 0',
	X =  118.374  mm,	Y =   -647.680  mm,	Z =   -250.000  mm,
	W =  90.000 deg,	P =   0.000 deg,	R =   90.000 deg
};
P[145]{
   GP1:
	UF : 0, UT : 6,		CONFIG : 'N U T, 0, 0, 0',
	X =  154.016  mm,	Y =   -627.100  mm,	Z =   -250.000  mm,
	W =  90.000 deg,	P =   0.000 deg,	R =   90.000 deg
};
P[146]{
   GP1:
	UF : 0, UT : 6,		CONFIG : 'N U T, 0, 0, 0',
	X =  189.658  mm,	Y =   -606.521  mm,	Z =   -250.000  mm,
	W =  90.000 deg,	P =   0.000 deg,	R =   90.000 deg
};
P[147]{
   GP1:
	UF : 0, UT : 6,		CONFIG : 'N U T, 0, 0, 0',
	X =  225.300  mm,	Y =   -585.941  mm,	Z =   -250.000  mm,
	W =  90.000 deg,	P =   0.000 deg,	R =   90.000 deg
};
P[148]{
   GP1:
	UF : 0, UT : 6,		CONFIG : 'N U T, 0, 0, 0',
	X =  260.942  mm,	Y =   -565.362  mm,	Z =   -250.000  mm,
	W =  90.000 deg,	P =   0.000 deg,	R =   90.000 deg
};
P[149]{
   GP1:
	UF : 0, UT : 6,		CONFIG : 'N U T, 0, 0, 0',
	X =  296.585  mm,	Y =   -544.783  mm,	Z =   -250.000  mm,
	W =  90.000 deg,	P =   0.000 deg,	R =   90.000 deg
};
P[150]{
   GP1:
	UF : 0, UT : 6,		CONFIG : 'N U T, 0, 0, 0',
	X =  332.227  mm,	Y =   -524.203  mm,	Z =   -250.000  mm,
	W =  90.000 deg,	P =   0.000 deg,	R =   90.000 deg
};
P[151]{
   GP1:
	UF : 0, UT : 6,		CONFIG : 'N U T, 0, 0, 0',
	X =  367.869  mm,	Y =   -503.624  mm,	Z =   -250.000  mm,
	W =  90.000 deg,	P =   0.000 deg,	R =   90.000 deg
};
P[152]{
   GP1:
	UF : 0, UT : 6,		CONFIG : 'N U T, 0, 0, 0',
	X =  403.511  mm,	Y =   -483.044  mm,	Z =   -250.000  mm,
	W =  90.000 deg,	P =   0.000 deg,	R =   90.000 deg
};
P[153]{
   GP1:
	UF : 0, UT : 6,		CONFIG : 'N U T, 0, 0, 0',
	X =  439.153  mm,	Y =   -462.465  mm,	Z =   -250.000  mm,
	W =  90.000 deg,	P =   0.000 deg,	R =   90.000 deg
};
P[154]{
   GP1:
	UF : 0, UT : 6,		CONFIG : 'N U T, 0, 0, 0',
	X =  474.795  mm,	Y =   -441.885  mm,	Z =   -250.000  mm,
	W =  90.000 deg,	P =   0.000 deg,	R =   90.000 deg
};
P[155]{
   GP1:
	UF : 0, UT : 6,		CONFIG : 'N U T, 0, 0, 0',
	X =  510.438  mm,	Y =   -421.306  mm,	Z =   -250.000  mm,
	W =  90.000 deg,	P =   0.000 deg,	R =   90.000 deg
};
P[156]{
   GP1:
	UF : 0, UT : 6,		CONFIG : 'N U T, 0, 0, 0',
	X =  195.000  mm,	Y =   -410.000  mm,	Z =   -170.000  mm,
	W =  90.000 deg,	P =   0.000 deg,	R =   90.000 deg
};
/END
